TYPE FB_ServoAchse_State :
(
	UNDEFINIERT := 0,
	STAND_BY,
	ENABLE,
	FAHRE_ABSOLUT,
	HAND,
	ERROR_HANDLER
);
END_TYPE

(* stored: Version 1.1.0.1, ProductVersion 3.1.4018.5
   DUT FB_ServoAchse_State: Id {54b96297-a0f8-45c5-8bb1-6a477800933c} *)
